{attribute 'qualified_only'}
VAR_GLOBAL CONSTANT
	  rMinWeightConstant : REAL  := 10.0;
      rMaxWeightConstant : REAL  := 550.0;
END_VAR

(* stored: Version 1.1.0.1, ProductVersion 3.1.4024.16
   GVL WeightConstants: Id {0b14448a-e6cf-4708-a448-b3d9c85f3c97} *)
